(* PLC project Generated.project, CODESYS CODESYS V3.5 SP19 Patch 1 *)
(* stored: creationDateTime 2026-09-06T13:00:42.404865, modificationDateTime 2026-09-06T13:00:42.404865 *)

(* values of E_MachineHomingStep: IDLE: Referencement indisponible (Enable=FALSE); LOSS_SAFESTOP: Perte de datum en mouvement : arret controle en cours; BOTH_NOT_HOMED: Codeurs M1 et M2 non references : passer en MAINT_N2; M1_NOT_HOMED: Codeur M1 non reference ou mesure douteuse : homer M1; M2_NOT_HOMED: Codeur M2 non reference ou mesure douteuse : homer M2; OFFSET_UNKNOWN: Offset benne inconnu : passer en MAINT_N2; NEED_TOP_POSITION: Monter Both a vitesse lente jusqu au capteur haut; NEED_MECHANICAL_STOP: Capteur haut atteint : relacher la commande et attendre l arret; AWAIT_BUCKET_CONFIRM: Confirmer visuellement la benne : Fermee ou Ouverte; HOMING_IN_PROGRESS: Referencement conjoint M1/M2 en cours : ne pas manoeuvrer; VALID: Referencement machine valide : mode nominal disponible; FAILED: Referencement incomplet : rester en N2 et recommencer *)

{attribute 'qualified_only'}
{attribute 'strict'}
TYPE E_MachineHomingStep : (IDLE := 0, LOSS_SAFESTOP := 5, BOTH_NOT_HOMED := 10, M1_NOT_HOMED := 11, M2_NOT_HOMED := 12, OFFSET_UNKNOWN := 20, NEED_TOP_POSITION := 30, NEED_MECHANICAL_STOP := 40, AWAIT_BUCKET_CONFIRM := 45, HOMING_IN_PROGRESS := 50, VALID := 60, FAILED := 70);
END_TYPE
